// Latched by the base on the Execute rising edge (S6.1).
TYPE ST_AxisParCmd :
STRUCT
    Target : LREAL;   // absolute target for MOVE_TO, in axis units
END_STRUCT
END_TYPE

(* stored: Version 1.1.0.1, ProductVersion 3.1.4024.12
   DUT ST_AxisParCmd: Id {e0eb10c1-5722-4d15-b626-177f132bbe7e} *)
